TYPE "A0301_Mach_Speed_Par"
VERSION : 0.1
// Block: A0301_Mach_Speed_Par
   STRUCT
      SemiAut_Vel : LReal;
      Aut_Vel : LReal;
      Aut_Acc : LReal;
      Aut_Dec : LReal;
   END_STRUCT;

END_TYPE
